TYPE E_MzHeaterType :
(
	Nothing,
	SingleHeater,	//MB
	TwinHeater,		//HT-Heater
	HeaterCooler	//Heizer und Kühler
);
END_TYPE

(* stored: Version 1.1.0.1, ProductVersion 3.1.4022.18
   DUT E_MzHeaterType: Id {adc18bf8-0b39-42e7-bb87-57adcbfb8708} *)
